(* IEC 61131-3 sources: CodesysTest/export/Function Blocks/FB_BaseObject.pou, 2 files *)

(* ---- FB_BaseObject.pou.st ---- *)
(*#-#-#-#-#-#-#-#-#-#---Declaration---#-#-#-#-#-#-#-#-#-#-#-#-#*)

FUNCTION_BLOCK FB_BaseObject IMPLEMENTS IAllObjects, ILoggable
VAR_INPUT
END_VAR
VAR_OUTPUT
END_VAR
VAR
	_instanceName : STRING;			// Instance Name
	_prefix : STRING;
	_logger : IMachineLogger;
END_VAR
(*#-#-#-#-#-#-#-#-#-#---Implementation---#-#-#-#-#-#-#-#-#-#-#-#-#*)

(* ---- FB_Init.m.st ---- *)
(*#-#-#-#-#-#-#-#-#-#---Declaration---#-#-#-#-#-#-#-#-#-#-#-#-#*)

METHOD FB_Init : BOOL
VAR_INPUT
  bInitRetains : BOOL; // TRUE: the retain variables are initialized (reset warm / reset cold)
  bInCopyCode : BOOL;  // TRUE: the instance will be copied to the copy code afterward (online change)
  name : STRING;
END_VAR
(*#-#-#-#-#-#-#-#-#-#---Implementation---#-#-#-#-#-#-#-#-#-#-#-#-#*)

_instanceName := name;
_prefix := CONCAT(name, ' ');
GlobalObjects.CollectionOfAllObjects.AddObject(THIS^);
